(* Logix 5000 project; controller TEC_81 vendor 1 type 14 code 148 rev 36.11; software revision 36.00; part 2 of 5 *)
(* tags used below, declared in another part *)
   B_Reset_Posicion_kinetix_0 : DINT;
   Ctrl_Kinetix_A1 : DINT;
   Done_Kinetx_0 : DINT;
   home_step_1 : BOOL;
   ok_com_1 : BOOL;
   reset_Kinetix_1 : BOOL;
   Axis_1 : AXIS_CIP_DRIVE;
   Axis_2 : AXIS_CIP_DRIVE;   // Almacen 2
   B_Reset_Posicion_kinetix : DINT;
   Ctrl_Kinetix_A2 : DINT;   // Boton Start Kinetix
   Done_Kinetx : DINT;
   Faul_Axis : DINT;
   In_Pos_Alm_2 : DINT;
   Kinetix_Pos_Alm_1 : DINT;
   Kinetix_Pos_Alm_2 : DINT;
   MAFR_Mtr_Alm_1 : MOTION_INSTRUCTION;
   MAFR_Mtr_Alm_2 : MOTION_INSTRUCTION;
   MAM_1_Mtr_Alm_0 : MOTION_INSTRUCTION;
   MAM_1_Mtr_Alm_1 : MOTION_INSTRUCTION;
   MAM_1_Mtr_Alm_2 : MOTION_INSTRUCTION;
   MAM_2_Mtr_Alm_1 : MOTION_INSTRUCTION;
   MAM_2_Mtr_Alm_2 : MOTION_INSTRUCTION;
   MAM_3_Mtr_Alm_1 : MOTION_INSTRUCTION;
   MAM_3_Mtr_Alm_2 : MOTION_INSTRUCTION;
   MAM_4_Mtr_Alm_1 : MOTION_INSTRUCTION;
   MAM_4_Mtr_Alm_2 : MOTION_INSTRUCTION;
   MAM_5_Mtr_Alm_1 : MOTION_INSTRUCTION;
   MAM_5_Mtr_Alm_2 : MOTION_INSTRUCTION;
   MAM_6_Mtr_Alm_1 : MOTION_INSTRUCTION;
   MAM_6_Mtr_Alm_2 : MOTION_INSTRUCTION;
   MAM_7_Mtr_Alm_2 : MOTION_INSTRUCTION;
   MAM_8_Mtr_Alm_1 : MOTION_INSTRUCTION;
   MAM_8_Mtr_Alm_2 : MOTION_INSTRUCTION;
   ok_com : BOOL;   // tag de prueba de comunicacion
   reset_Kinetix : BOOL;
   servo_start : MOTION_INSTRUCTION;
   servo_start_01 : MOTION_INSTRUCTION;
   Sevo_Stop : MOTION_INSTRUCTION;
   Start_Kinetix_Alm_2 : DINT;
   To_Pos_Alm_1 : DINT;
   To_Pos_Alm_2 : DINT;
(* _Almacen_1, continued *)

ROUTINE Start_KInetixA1   (* ladder *)
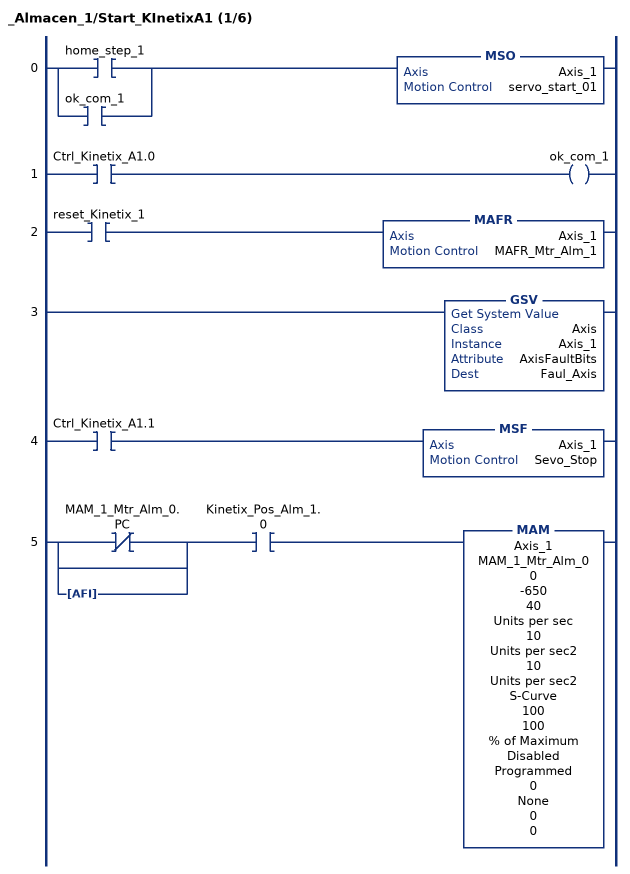
   0: [XIC(home_step_1) ,XIC(ok_com_1) ]MSO(Axis_1,servo_start_01);
   1: XIC(Ctrl_Kinetix_A1.0)OTE(ok_com_1);
   2: XIC(reset_Kinetix_1)MAFR(Axis_1,MAFR_Mtr_Alm_1);
   3: GSV(Axis,Axis_1,AxisFaultBits,Faul_Axis);
   4: XIC(Ctrl_Kinetix_A1.1)MSF(Axis_1,Sevo_Stop);
   5: [XIO(MAM_1_Mtr_Alm_0.PC) ,,AFI() ]XIC(Kinetix_Pos_Alm_1.0)MAM(Axis_1,MAM_1_Mtr_Alm_0,0,-650,40,Units per sec,10,Units per sec2,10,Units per sec2,S-Curve,100,100,% of Maximum,Disabled,Programmed,0,None,0,0);
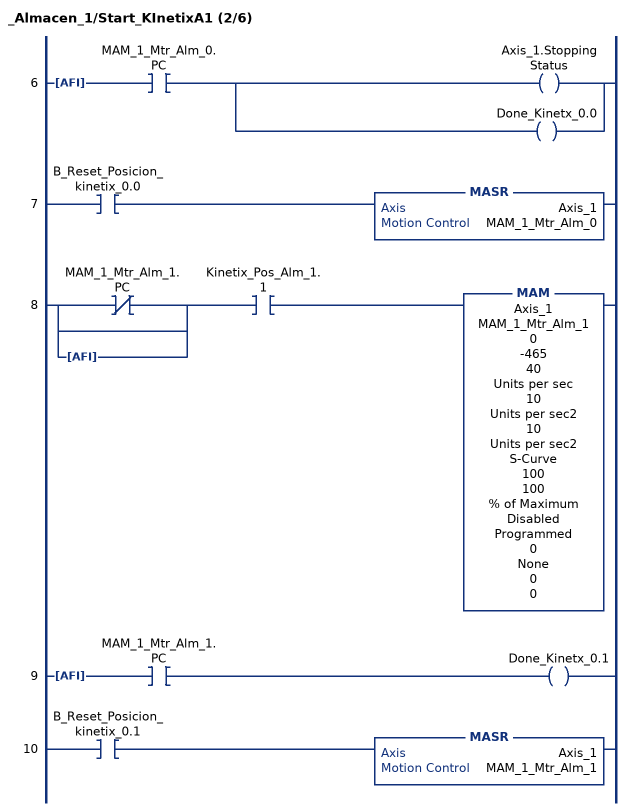
   6: AFI()XIC(MAM_1_Mtr_Alm_0.PC)[OTE(Axis_1.StoppingStatus) ,OTE(Done_Kinetx_0.0) ];
   7: XIC(B_Reset_Posicion_kinetix_0.0)MASR(Axis_1,MAM_1_Mtr_Alm_0);
   8: [XIO(MAM_1_Mtr_Alm_1.PC) ,,AFI() ]XIC(Kinetix_Pos_Alm_1.1)MAM(Axis_1,MAM_1_Mtr_Alm_1,0,-465,40,Units per sec,10,Units per sec2,10,Units per sec2,S-Curve,100,100,% of Maximum,Disabled,Programmed,0,None,0,0);
   9: AFI()XIC(MAM_1_Mtr_Alm_1.PC)OTE(Done_Kinetx_0.1);
   10: XIC(B_Reset_Posicion_kinetix_0.1)MASR(Axis_1,MAM_1_Mtr_Alm_1);
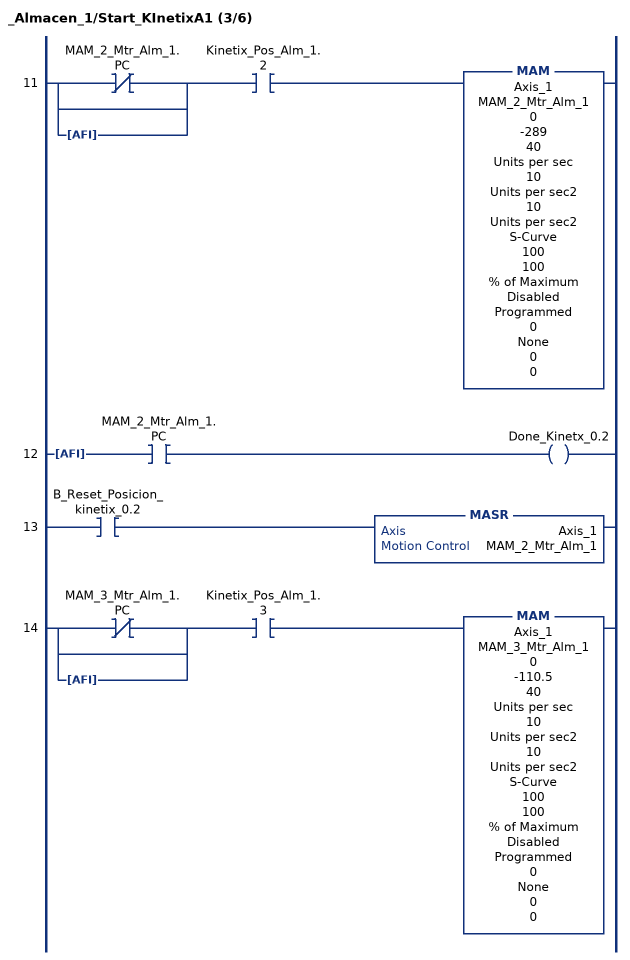
   11: [XIO(MAM_2_Mtr_Alm_1.PC) ,,AFI() ]XIC(Kinetix_Pos_Alm_1.2)MAM(Axis_1,MAM_2_Mtr_Alm_1,0,-289,40,Units per sec,10,Units per sec2,10,Units per sec2,S-Curve,100,100,% of Maximum,Disabled,Programmed,0,None,0,0);
   12: AFI()XIC(MAM_2_Mtr_Alm_1.PC)OTE(Done_Kinetx_0.2);
   13: XIC(B_Reset_Posicion_kinetix_0.2)MASR(Axis_1,MAM_2_Mtr_Alm_1);
   14: [XIO(MAM_3_Mtr_Alm_1.PC) ,,AFI() ]XIC(Kinetix_Pos_Alm_1.3)MAM(Axis_1,MAM_3_Mtr_Alm_1,0,-110.5,40,Units per sec,10,Units per sec2,10,Units per sec2,S-Curve,100,100,% of Maximum,Disabled,Programmed,0,None,0,0);
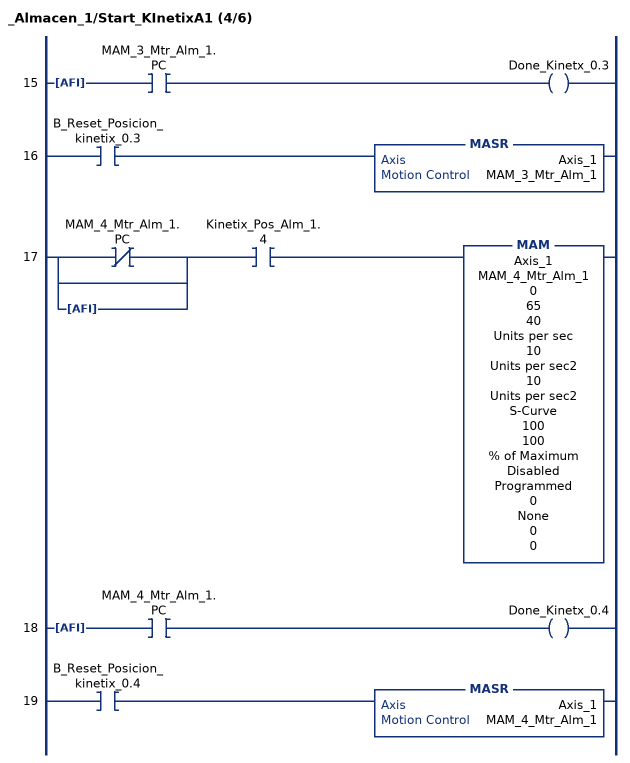
   15: AFI()XIC(MAM_3_Mtr_Alm_1.PC)OTE(Done_Kinetx_0.3);
   16: XIC(B_Reset_Posicion_kinetix_0.3)MASR(Axis_1,MAM_3_Mtr_Alm_1);
   17: [XIO(MAM_4_Mtr_Alm_1.PC) ,,AFI() ]XIC(Kinetix_Pos_Alm_1.4)MAM(Axis_1,MAM_4_Mtr_Alm_1,0,65,40,Units per sec,10,Units per sec2,10,Units per sec2,S-Curve,100,100,% of Maximum,Disabled,Programmed,0,None,0,0);
   18: AFI()XIC(MAM_4_Mtr_Alm_1.PC)OTE(Done_Kinetx_0.4);
   19: XIC(B_Reset_Posicion_kinetix_0.4)MASR(Axis_1,MAM_4_Mtr_Alm_1);
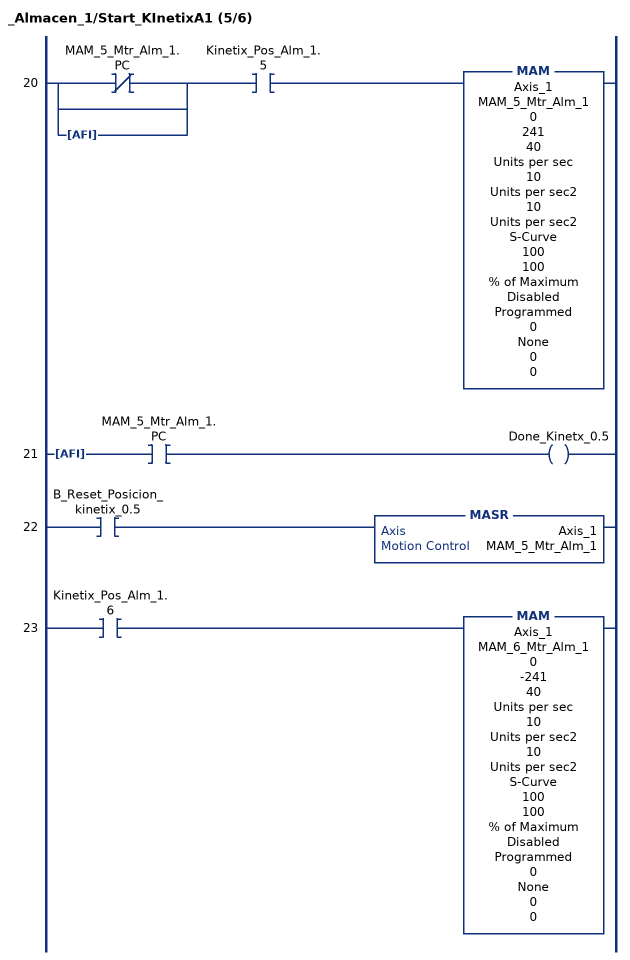
   20: [XIO(MAM_5_Mtr_Alm_1.PC) ,,AFI() ]XIC(Kinetix_Pos_Alm_1.5)MAM(Axis_1,MAM_5_Mtr_Alm_1,0,241,40,Units per sec,10,Units per sec2,10,Units per sec2,S-Curve,100,100,% of Maximum,Disabled,Programmed,0,None,0,0);
   21: AFI()XIC(MAM_5_Mtr_Alm_1.PC)OTE(Done_Kinetx_0.5);
   22: XIC(B_Reset_Posicion_kinetix_0.5)MASR(Axis_1,MAM_5_Mtr_Alm_1);
   23: XIC(Kinetix_Pos_Alm_1.6)MAM(Axis_1,MAM_6_Mtr_Alm_1,0,-241,40,Units per sec,10,Units per sec2,10,Units per sec2,S-Curve,100,100,% of Maximum,Disabled,Programmed,0,None,0,0);
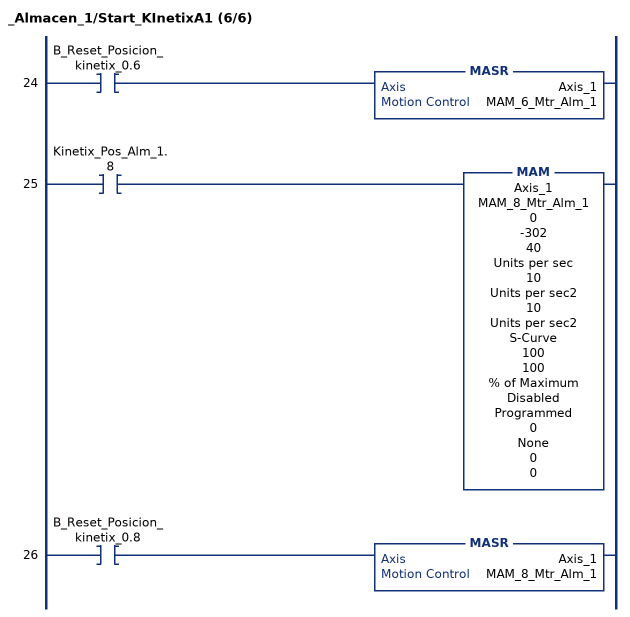
   24: XIC(B_Reset_Posicion_kinetix_0.6)MASR(Axis_1,MAM_6_Mtr_Alm_1);
   25: XIC(Kinetix_Pos_Alm_1.8)MAM(Axis_1,MAM_8_Mtr_Alm_1,0,-302,40,Units per sec,10,Units per sec2,10,Units per sec2,S-Curve,100,100,% of Maximum,Disabled,Programmed,0,None,0,0);
   26: XIC(B_Reset_Posicion_kinetix_0.8)MASR(Axis_1,MAM_8_Mtr_Alm_1);
END_ROUTINE
END_PROGRAM

PROGRAM _Almacen_2   (* main routine _01_Main *)
VAR
   home_step : BOOL;
END_VAR

ROUTINE _01_Main   (* ladder *)
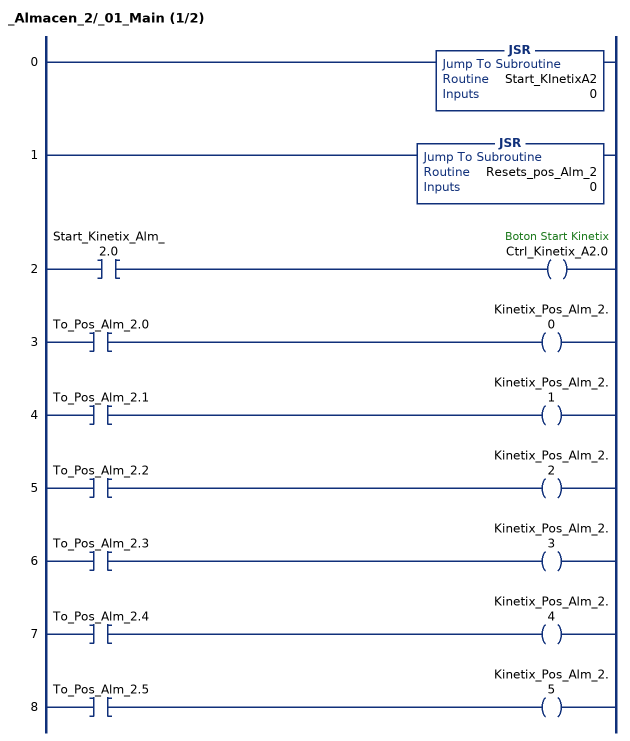
   0: JSR(Start_KInetixA2,0);
   1: JSR(Resets_pos_Alm_2,0);
   2: XIC(Start_Kinetix_Alm_2.0)OTE(Ctrl_Kinetix_A2.0);
   3: XIC(To_Pos_Alm_2.0)OTE(Kinetix_Pos_Alm_2.0);
   4: XIC(To_Pos_Alm_2.1)OTE(Kinetix_Pos_Alm_2.1);
   5: XIC(To_Pos_Alm_2.2)OTE(Kinetix_Pos_Alm_2.2);
   6: XIC(To_Pos_Alm_2.3)OTE(Kinetix_Pos_Alm_2.3);
   7: XIC(To_Pos_Alm_2.4)OTE(Kinetix_Pos_Alm_2.4);
   8: XIC(To_Pos_Alm_2.5)OTE(Kinetix_Pos_Alm_2.5);
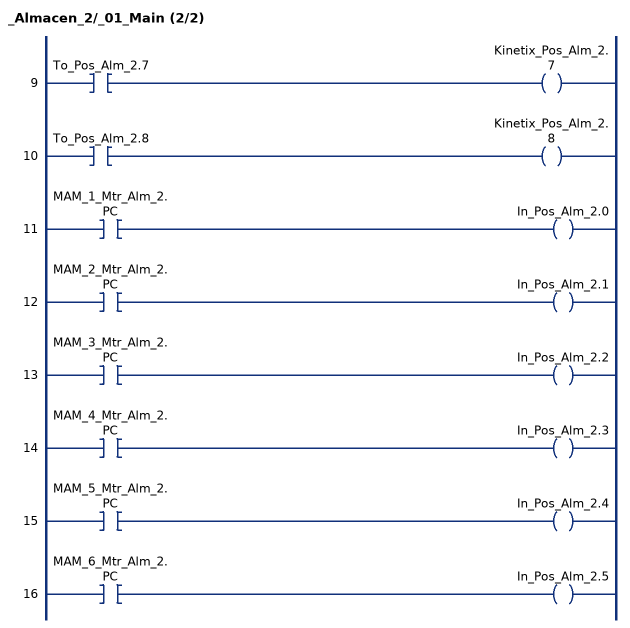
   9: XIC(To_Pos_Alm_2.7)OTE(Kinetix_Pos_Alm_2.7);
   10: XIC(To_Pos_Alm_2.8)OTE(Kinetix_Pos_Alm_2.8);
   11: XIC(MAM_1_Mtr_Alm_2.PC)OTE(In_Pos_Alm_2.0);
   12: XIC(MAM_2_Mtr_Alm_2.PC)OTE(In_Pos_Alm_2.1);
   13: XIC(MAM_3_Mtr_Alm_2.PC)OTE(In_Pos_Alm_2.2);
   14: XIC(MAM_4_Mtr_Alm_2.PC)OTE(In_Pos_Alm_2.3);
   15: XIC(MAM_5_Mtr_Alm_2.PC)OTE(In_Pos_Alm_2.4);
   16: XIC(MAM_6_Mtr_Alm_2.PC)OTE(In_Pos_Alm_2.5);
END_ROUTINE

ROUTINE Resets_pos_Alm_2   (* ladder *)
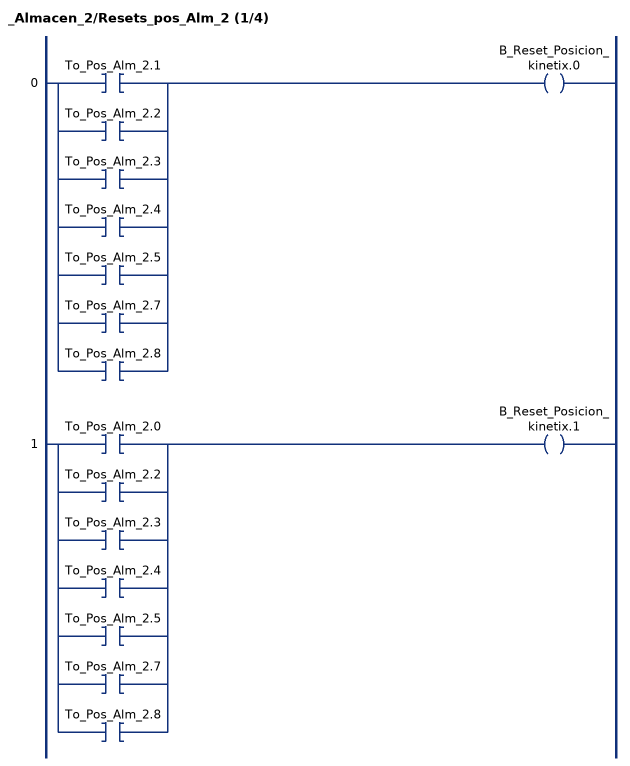
   0: [XIC(To_Pos_Alm_2.1) ,XIC(To_Pos_Alm_2.2) ,XIC(To_Pos_Alm_2.3) ,XIC(To_Pos_Alm_2.4) ,XIC(To_Pos_Alm_2.5) ,XIC(To_Pos_Alm_2.7) ,XIC(To_Pos_Alm_2.8) ]OTE(B_Reset_Posicion_kinetix.0);
   1: [XIC(To_Pos_Alm_2.0) ,XIC(To_Pos_Alm_2.2) ,XIC(To_Pos_Alm_2.3) ,XIC(To_Pos_Alm_2.4) ,XIC(To_Pos_Alm_2.5) ,XIC(To_Pos_Alm_2.7) ,XIC(To_Pos_Alm_2.8) ]OTE(B_Reset_Posicion_kinetix.1);
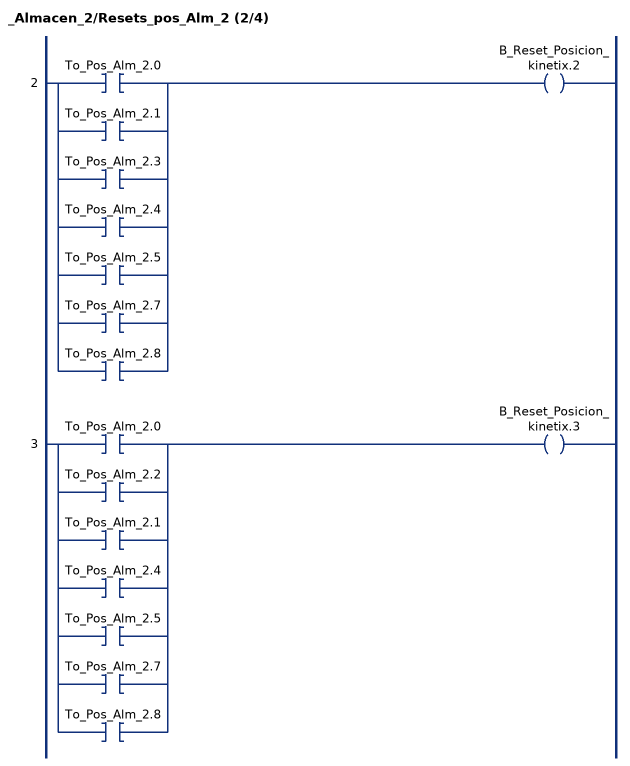
   2: [XIC(To_Pos_Alm_2.0) ,XIC(To_Pos_Alm_2.1) ,XIC(To_Pos_Alm_2.3) ,XIC(To_Pos_Alm_2.4) ,XIC(To_Pos_Alm_2.5) ,XIC(To_Pos_Alm_2.7) ,XIC(To_Pos_Alm_2.8) ]OTE(B_Reset_Posicion_kinetix.2);
   3: [XIC(To_Pos_Alm_2.0) ,XIC(To_Pos_Alm_2.2) ,XIC(To_Pos_Alm_2.1) ,XIC(To_Pos_Alm_2.4) ,XIC(To_Pos_Alm_2.5) ,XIC(To_Pos_Alm_2.7) ,XIC(To_Pos_Alm_2.8) ]OTE(B_Reset_Posicion_kinetix.3);
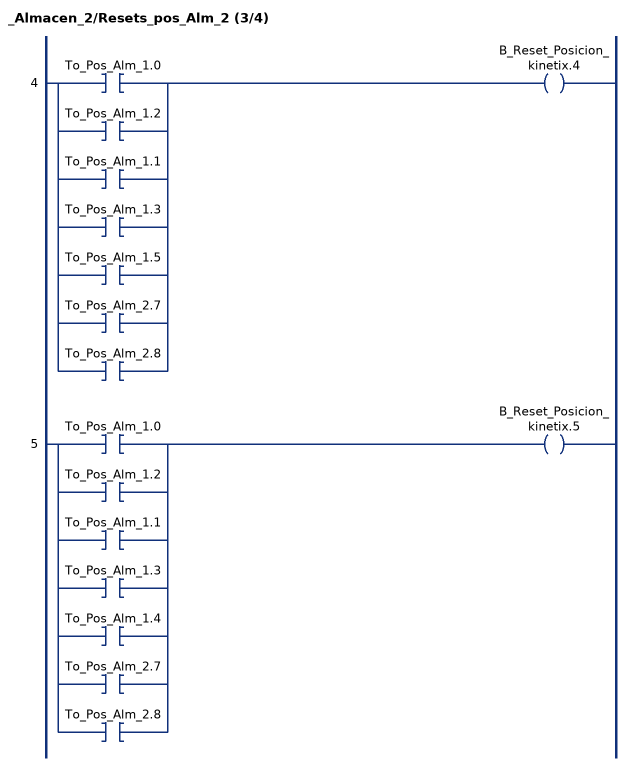
   4: [XIC(To_Pos_Alm_1.0) ,XIC(To_Pos_Alm_1.2) ,XIC(To_Pos_Alm_1.1) ,XIC(To_Pos_Alm_1.3) ,XIC(To_Pos_Alm_1.5) ,XIC(To_Pos_Alm_2.7) ,XIC(To_Pos_Alm_2.8) ]OTE(B_Reset_Posicion_kinetix.4);
   5: [XIC(To_Pos_Alm_1.0) ,XIC(To_Pos_Alm_1.2) ,XIC(To_Pos_Alm_1.1) ,XIC(To_Pos_Alm_1.3) ,XIC(To_Pos_Alm_1.4) ,XIC(To_Pos_Alm_2.7) ,XIC(To_Pos_Alm_2.8) ]OTE(B_Reset_Posicion_kinetix.5);
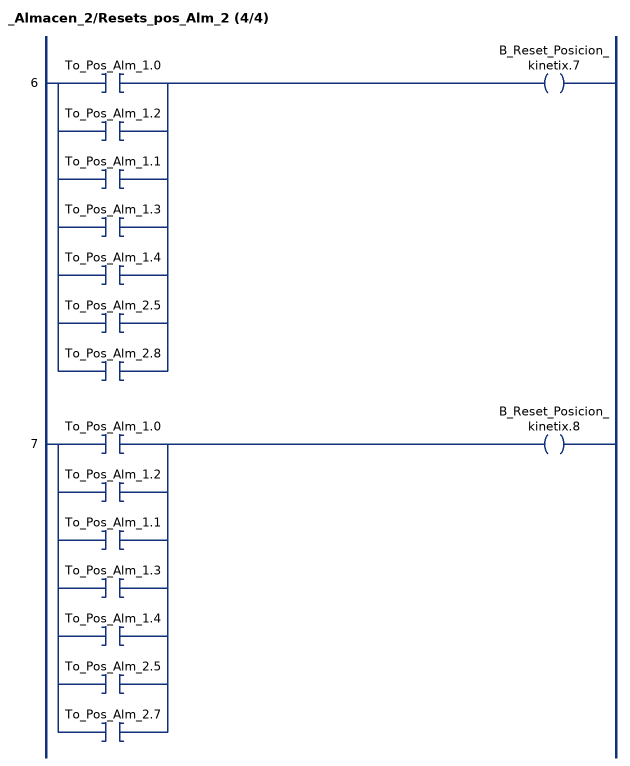
   6: [XIC(To_Pos_Alm_1.0) ,XIC(To_Pos_Alm_1.2) ,XIC(To_Pos_Alm_1.1) ,XIC(To_Pos_Alm_1.3) ,XIC(To_Pos_Alm_1.4) ,XIC(To_Pos_Alm_2.5) ,XIC(To_Pos_Alm_2.8) ]OTE(B_Reset_Posicion_kinetix.7);
   7: [XIC(To_Pos_Alm_1.0) ,XIC(To_Pos_Alm_1.2) ,XIC(To_Pos_Alm_1.1) ,XIC(To_Pos_Alm_1.3) ,XIC(To_Pos_Alm_1.4) ,XIC(To_Pos_Alm_2.5) ,XIC(To_Pos_Alm_2.7) ]OTE(B_Reset_Posicion_kinetix.8);
END_ROUTINE

ROUTINE Start_KInetixA2   (* ladder *)
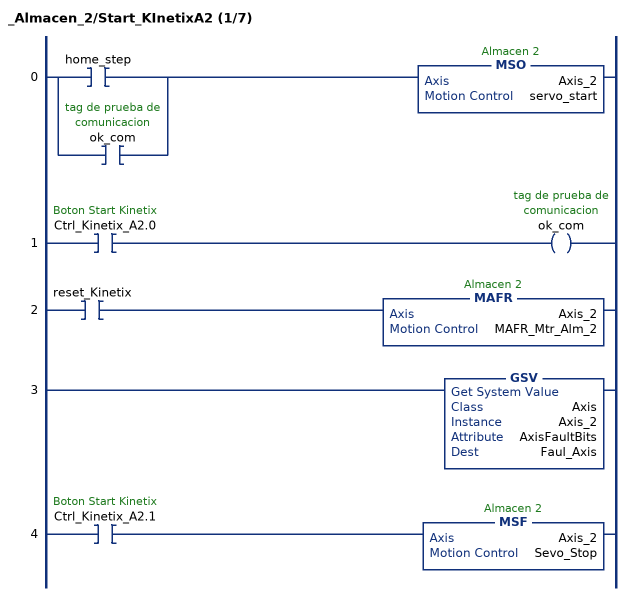
   0: [XIC(home_step) ,XIC(ok_com) ]MSO(Axis_2,servo_start);
   1: XIC(Ctrl_Kinetix_A2.0)OTE(ok_com);
   2: XIC(reset_Kinetix)MAFR(Axis_2,MAFR_Mtr_Alm_2);
   3: GSV(Axis,Axis_2,AxisFaultBits,Faul_Axis);
   4: XIC(Ctrl_Kinetix_A2.1)MSF(Axis_2,Sevo_Stop);
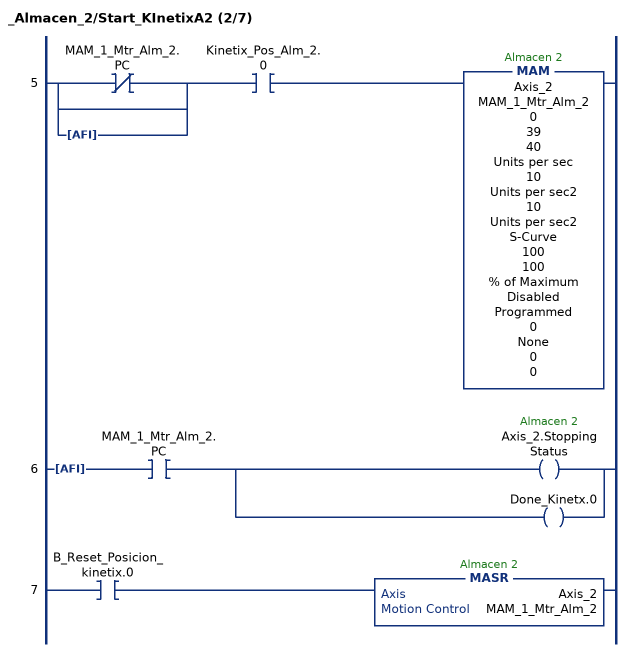
   5: [XIO(MAM_1_Mtr_Alm_2.PC) ,,AFI() ]XIC(Kinetix_Pos_Alm_2.0)MAM(Axis_2,MAM_1_Mtr_Alm_2,0,39,40,Units per sec,10,Units per sec2,10,Units per sec2,S-Curve,100,100,% of Maximum,Disabled,Programmed,0,None,0,0);
   6: AFI()XIC(MAM_1_Mtr_Alm_2.PC)[OTE(Axis_2.StoppingStatus) ,OTE(Done_Kinetx.0) ];
   7: XIC(B_Reset_Posicion_kinetix.0)MASR(Axis_2,MAM_1_Mtr_Alm_2);
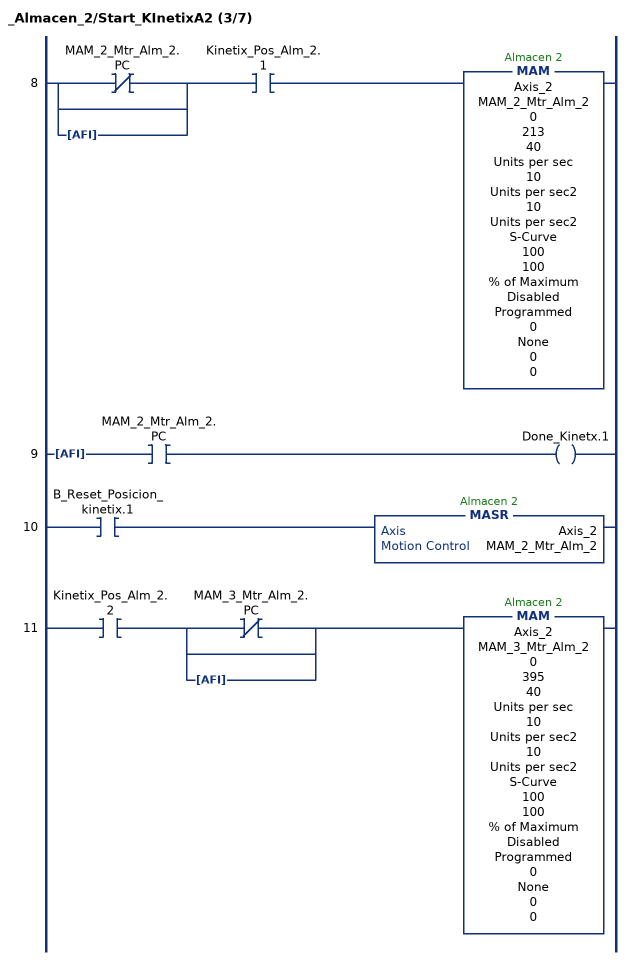
   8: [XIO(MAM_2_Mtr_Alm_2.PC) ,,AFI() ]XIC(Kinetix_Pos_Alm_2.1)MAM(Axis_2,MAM_2_Mtr_Alm_2,0,213,40,Units per sec,10,Units per sec2,10,Units per sec2,S-Curve,100,100,% of Maximum,Disabled,Programmed,0,None,0,0);
   9: AFI()XIC(MAM_2_Mtr_Alm_2.PC)OTE(Done_Kinetx.1);
   10: XIC(B_Reset_Posicion_kinetix.1)MASR(Axis_2,MAM_2_Mtr_Alm_2);
   11: XIC(Kinetix_Pos_Alm_2.2)[XIO(MAM_3_Mtr_Alm_2.PC) ,,AFI() ]MAM(Axis_2,MAM_3_Mtr_Alm_2,0,395,40,Units per sec,10,Units per sec2,10,Units per sec2,S-Curve,100,100,% of Maximum,Disabled,Programmed,0,None,0,0);
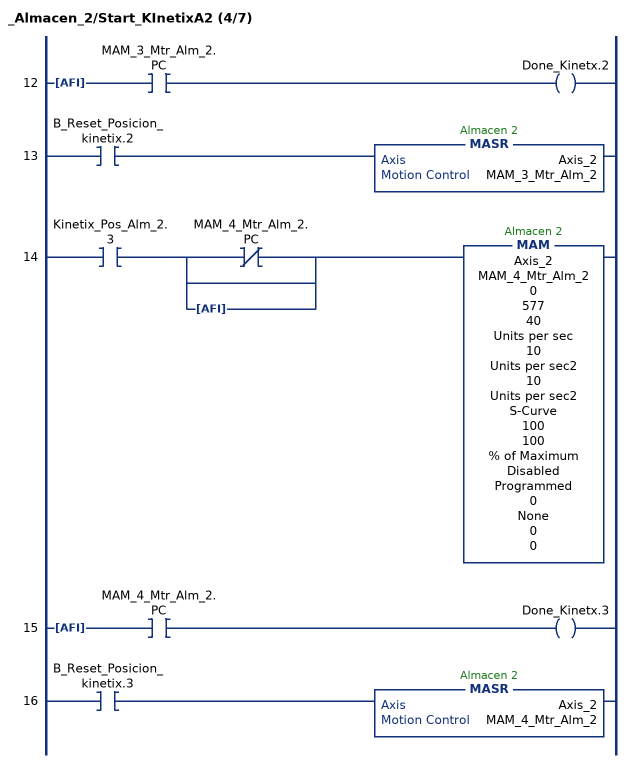
   12: AFI()XIC(MAM_3_Mtr_Alm_2.PC)OTE(Done_Kinetx.2);
   13: XIC(B_Reset_Posicion_kinetix.2)MASR(Axis_2,MAM_3_Mtr_Alm_2);
   14: XIC(Kinetix_Pos_Alm_2.3)[XIO(MAM_4_Mtr_Alm_2.PC) ,,AFI() ]MAM(Axis_2,MAM_4_Mtr_Alm_2,0,577,40,Units per sec,10,Units per sec2,10,Units per sec2,S-Curve,100,100,% of Maximum,Disabled,Programmed,0,None,0,0);
   15: AFI()XIC(MAM_4_Mtr_Alm_2.PC)OTE(Done_Kinetx.3);
   16: XIC(B_Reset_Posicion_kinetix.3)MASR(Axis_2,MAM_4_Mtr_Alm_2);
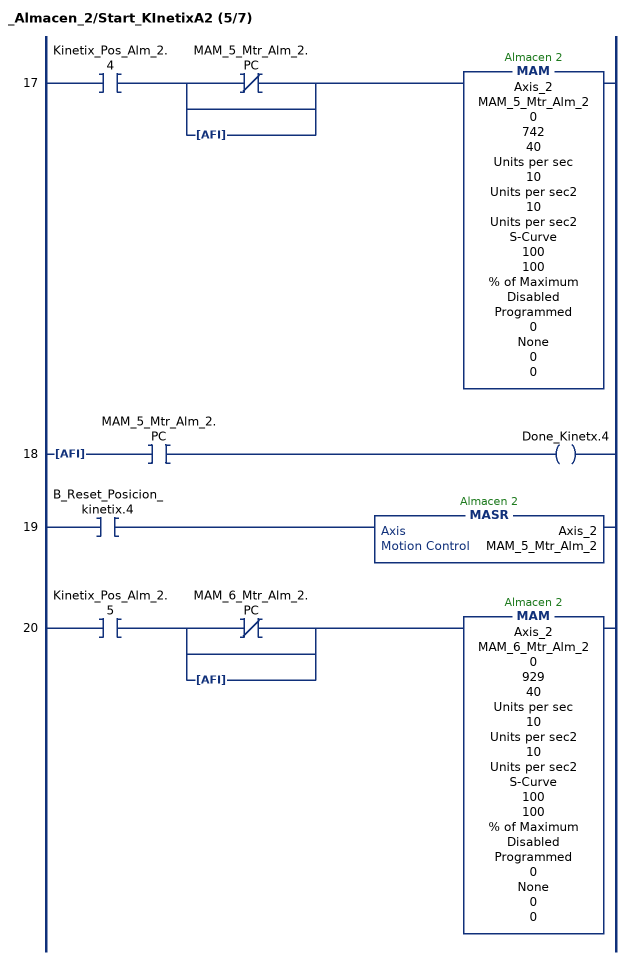
   17: XIC(Kinetix_Pos_Alm_2.4)[XIO(MAM_5_Mtr_Alm_2.PC) ,,AFI() ]MAM(Axis_2,MAM_5_Mtr_Alm_2,0,742,40,Units per sec,10,Units per sec2,10,Units per sec2,S-Curve,100,100,% of Maximum,Disabled,Programmed,0,None,0,0);
   18: AFI()XIC(MAM_5_Mtr_Alm_2.PC)OTE(Done_Kinetx.4);
   19: XIC(B_Reset_Posicion_kinetix.4)MASR(Axis_2,MAM_5_Mtr_Alm_2);
   20: XIC(Kinetix_Pos_Alm_2.5)[XIO(MAM_6_Mtr_Alm_2.PC) ,,AFI() ]MAM(Axis_2,MAM_6_Mtr_Alm_2,0,929,40,Units per sec,10,Units per sec2,10,Units per sec2,S-Curve,100,100,% of Maximum,Disabled,Programmed,0,None,0,0);
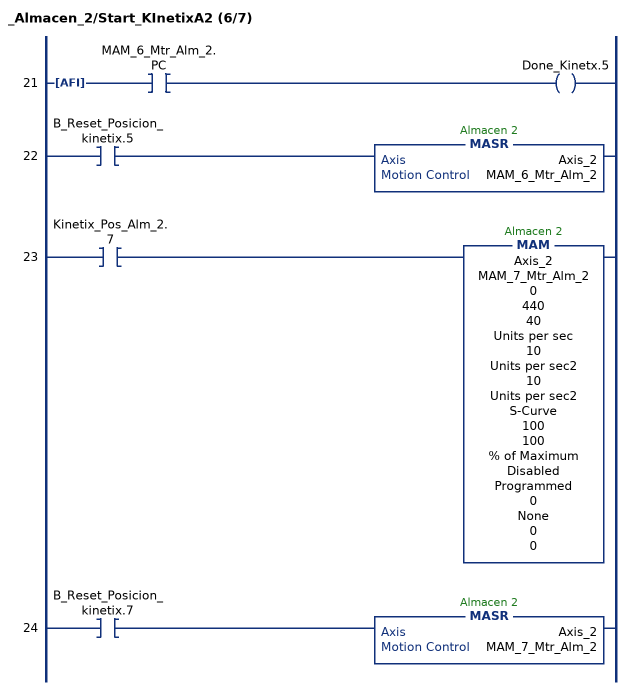
   21: AFI()XIC(MAM_6_Mtr_Alm_2.PC)OTE(Done_Kinetx.5);
   22: XIC(B_Reset_Posicion_kinetix.5)MASR(Axis_2,MAM_6_Mtr_Alm_2);
   23: XIC(Kinetix_Pos_Alm_2.7)MAM(Axis_2,MAM_7_Mtr_Alm_2,0,440,40,Units per sec,10,Units per sec2,10,Units per sec2,S-Curve,100,100,% of Maximum,Disabled,Programmed,0,None,0,0);
   24: XIC(B_Reset_Posicion_kinetix.7)MASR(Axis_2,MAM_7_Mtr_Alm_2);
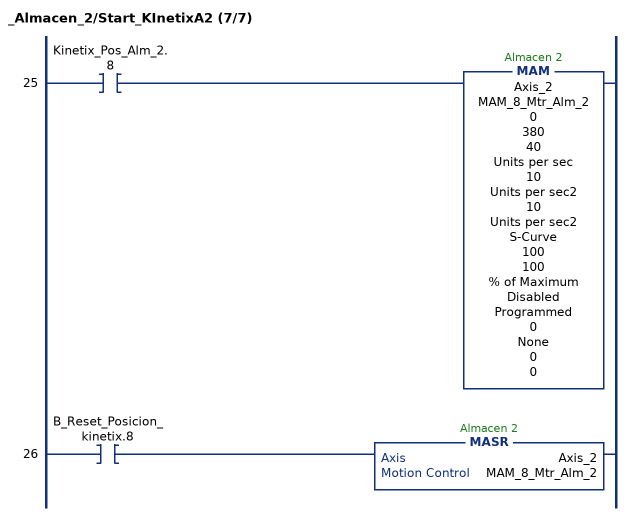
   25: XIC(Kinetix_Pos_Alm_2.8)MAM(Axis_2,MAM_8_Mtr_Alm_2,0,380,40,Units per sec,10,Units per sec2,10,Units per sec2,S-Curve,100,100,% of Maximum,Disabled,Programmed,0,None,0,0);
   26: XIC(B_Reset_Posicion_kinetix.8)MASR(Axis_2,MAM_8_Mtr_Alm_2);
END_ROUTINE
END_PROGRAM
